# EPICS autosave request: iocs/scanSimIOC/iocBoot/iocScanSim/auto_settings.req
file "ADDRIVERNAMESTANDARD_settings.req",  P=$(P),  R=cam1:
file "NDStdArrays_settings.req",  P=$(P),  R=image1:
file "commonPlugin_settings.req", P=$(P)
